DATA_BLOCK "BlockIncrementer_DB"
{ S7_Optimized_Access := 'TRUE' }
VERSION : 0.1
NON_RETAIN
"BlockIncrementer"

BEGIN

END_DATA_BLOCK

